PROGRAM ControlLD
VAR
	Ready: RS;
	level1: RS;
	L1toL3: RS;
	Level3: RS;
	L3ToL1: RS;
	L1toL2: RS;
	L3toL2: RS;
	Level2: RS;
	L2toL1: RS;
	L2toL3: RS;
	MotorUpTimerr: TON;
	MotorDownTimerr: TON;
END_VAR
VAR // added by the converter: edge detectors and wires of the graphical bodies
    _w1, _w2, _w3 : BOOL;
END_VAR

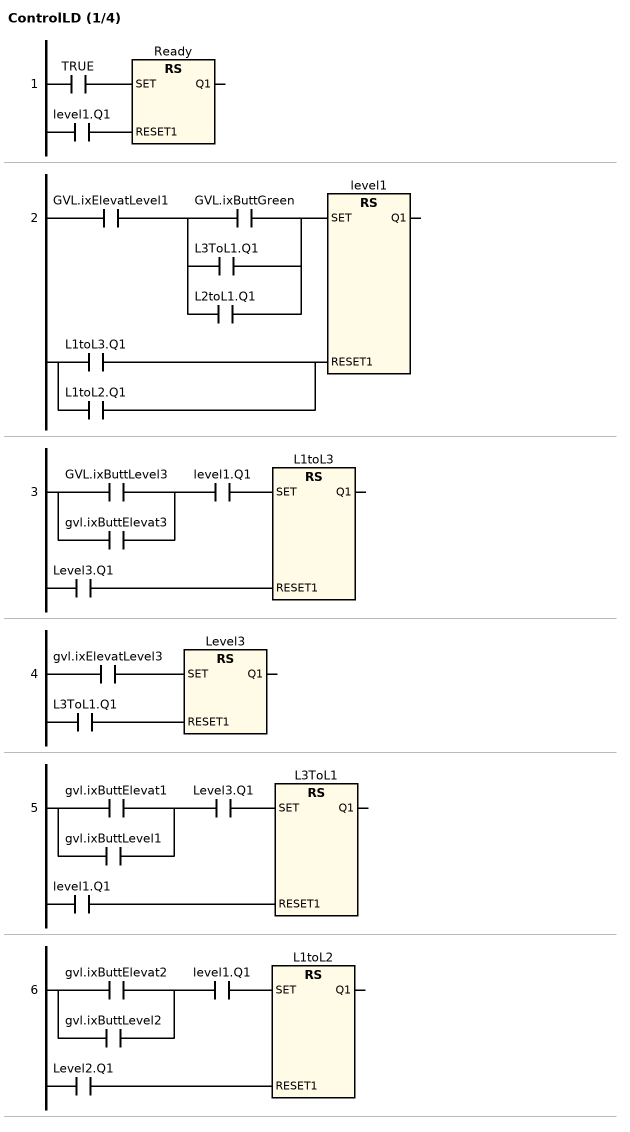
// NETWORK 1
Ready(SET := TRUE, RESET1 := level1.Q1); // RS

// NETWORK 2
level1(SET := GVL.ixElevatLevel1 AND (GVL.ixButtGreen OR L3ToL1.Q1 OR L2toL1.Q1), RESET1 := L1toL3.Q1 OR L1toL2.Q1); // RS

// NETWORK 3
L1toL3(SET := (GVL.ixButtLevel3 OR gvl.ixButtElevat3) AND level1.Q1, RESET1 := Level3.Q1); // RS

// NETWORK 4
Level3(SET := gvl.ixElevatLevel3, RESET1 := L3ToL1.Q1); // RS

// NETWORK 5
L3ToL1(SET := (gvl.ixButtElevat1 OR gvl.ixButtLevel1) AND Level3.Q1, RESET1 := level1.Q1); // RS

// NETWORK 6
L1toL2(SET := (gvl.ixButtElevat2 OR gvl.ixButtLevel2) AND level1.Q1, RESET1 := Level2.Q1); // RS

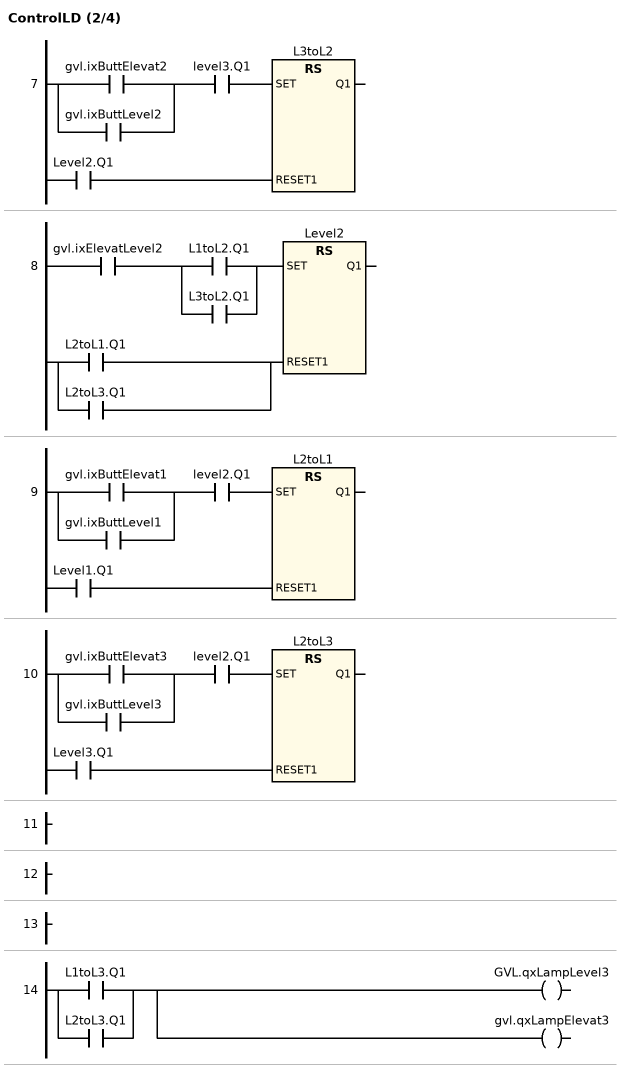
// NETWORK 7
L3toL2(SET := (gvl.ixButtElevat2 OR gvl.ixButtLevel2) AND level3.Q1, RESET1 := Level2.Q1); // RS

// NETWORK 8
Level2(SET := gvl.ixElevatLevel2 AND (L1toL2.Q1 OR L3toL2.Q1), RESET1 := L2toL1.Q1 OR L2toL3.Q1); // RS

// NETWORK 9
L2toL1(SET := (gvl.ixButtElevat1 OR gvl.ixButtLevel1) AND level2.Q1, RESET1 := Level1.Q1); // RS

// NETWORK 10
L2toL3(SET := (gvl.ixButtElevat3 OR gvl.ixButtLevel3) AND level2.Q1, RESET1 := Level3.Q1); // RS

// NETWORK 11

// NETWORK 12

// NETWORK 13

// NETWORK 14
_w1 := L1toL3.Q1 OR L2toL3.Q1;
GVL.qxLampLevel3 := _w1;
gvl.qxLampElevat3 := _w1;

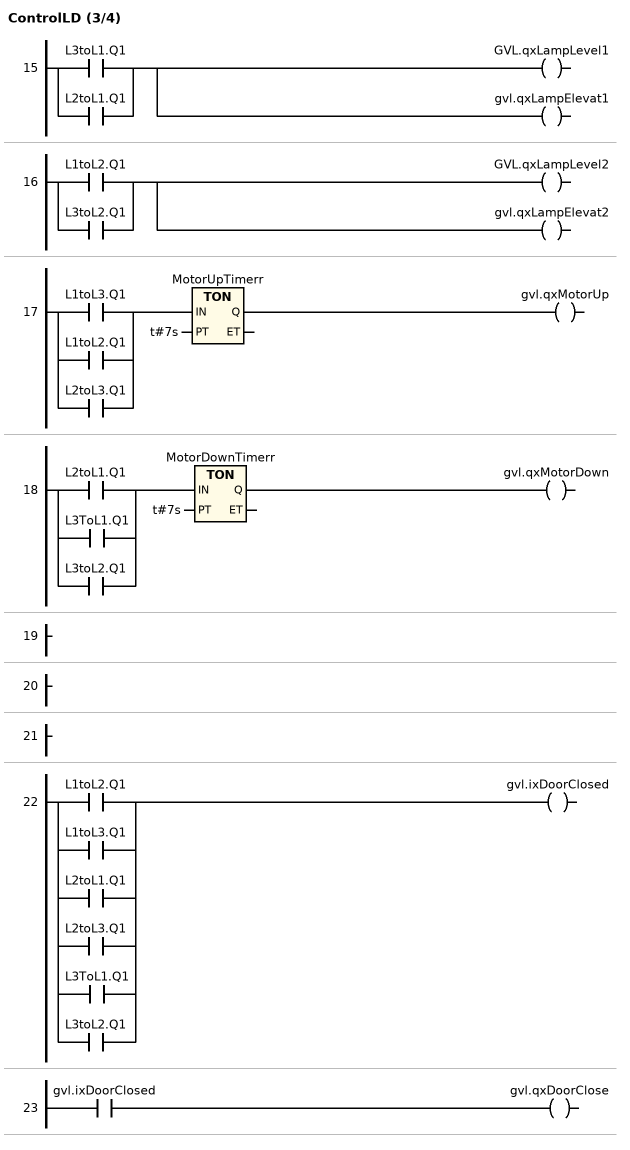
// NETWORK 15
_w2 := L3toL1.Q1 OR L2toL1.Q1;
GVL.qxLampLevel1 := _w2;
gvl.qxLampElevat1 := _w2;

// NETWORK 16
_w3 := L1toL2.Q1 OR L3toL2.Q1;
GVL.qxLampLevel2 := _w3;
gvl.qxLampElevat2 := _w3;

// NETWORK 17
MotorUpTimerr(IN := L1toL3.Q1 OR L1toL2.Q1 OR L2toL3.Q1, PT := t#7s); // TON
gvl.qxMotorUp := MotorUpTimerr.Q;

// NETWORK 18
MotorDownTimerr(IN := L2toL1.Q1 OR L3ToL1.Q1 OR L3toL2.Q1, PT := t#7s); // TON
gvl.qxMotorDown := MotorDownTimerr.Q;

// NETWORK 19

// NETWORK 20

// NETWORK 21

// NETWORK 22
gvl.ixDoorClosed := L1toL2.Q1 OR L1toL3.Q1 OR L2toL1.Q1 OR L2toL3.Q1 OR L3ToL1.Q1 OR L3toL2.Q1;

// NETWORK 23
gvl.qxDoorClose := gvl.ixDoorClosed;

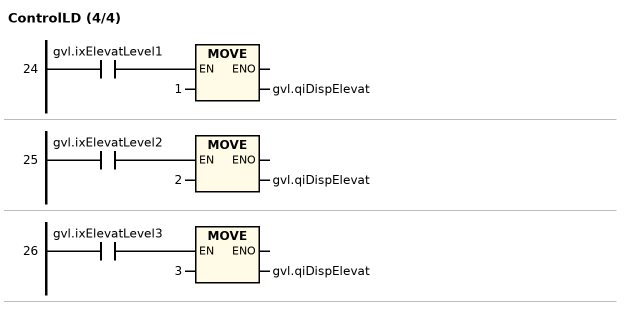
// NETWORK 24
IF gvl.ixElevatLevel1 THEN gvl.qiDispElevat := 1; END_IF

// NETWORK 25
IF gvl.ixElevatLevel2 THEN gvl.qiDispElevat := 2; END_IF

// NETWORK 26
IF gvl.ixElevatLevel3 THEN gvl.qiDispElevat := 3; END_IF

END_PROGRAM

(* stored: Version 1.1.0.1, ProductVersion 3.1.4024.12
   POU ControlLD: Id {912119c4-f197-4ac1-96d5-56b57bc2b241}, SpecialFunc None *)
